//{attribute 'qualified_only'}
VAR_GLOBAL
    (*DP1 ISOLATION VALVE*)
    {attribute 'TcLinkTo' := 	'.i_xOpnLS	:=	TIIB[K4S8_DRL_03_E10_EL1004]^Channel 1^Input;
                                 .i_xClsLS	:=	TIIB[K4S8_DRL_03_E10_EL1004]^Channel 2^Input;
                                 .q_xOPN_DO	:=	TIIB[K4S8_DRL_03_E11_EL2004]^Channel 2^Output
    '}
    {attribute 'pytmc' :=' pv: DREAM:DP1:VRC:01'}
    DREAM_DP1_VRC_01: FB_VRC;

    {attribute 'TcLinkTo' := 	'.i_xOpnLS	:=	TIIB[K4S8_DRL_03_E10_EL1004]^Channel 3^Input;
                                 .i_xClsLS	:=	TIIB[K4S8_DRL_03_E10_EL1004]^Channel 4^Input;
                                 .q_xCLS_DO	:=	TIIB[K4S8_DRL_03_E11_EL2004]^Channel 1^Output
    '}
    {attribute 'pytmc' :=' pv: DREAM:DP1:VRC:02'}
    DREAM_DP1_VRC_02: FB_VRC_NO;

    (*CATCHER 1 ISOLATION VALVE*)
    {attribute 'TcLinkTo' := 	'.i_xOpnLS	:=	TIIB[K4S8_DRL_04_E1_EL1004]^Channel 1^Input;
                                 .i_xClsLS	:=	TIIB[K4S8_DRL_04_E1_EL1004]^Channel 2^Input;
                                 .q_xOPN_DO	:=	TIIB[K4S8_DRL_04_E2_EL2004]^Channel 1^Output
    '}
    {attribute 'pytmc' :=' pv: DREAM:CAT1:VRC:01'}
    DREAM_CAT1_VRC_01: FB_VRC;

    (*ANGLE VALVES ROUGHING*)
    //Pneumatic valves
    {attribute 'TcLinkTo' := 	'.i_xOpnLS	:=	TIIB[K4S8_DRL_04_E9_EL1004]^Channel 1^Input;
                                 .i_xClsLS	:=	TIIB[K4S8_DRL_04_E9_EL1004]^Channel 2^Input;
                                 .q_xOPN_DO	:=	TIIB[K4S8_DRL_04_E11_EL2004]^Channel 1^Output
    '}
    {attribute 'pytmc' :=' pv: DREAM:ROUGH1:VRC:01'}
    DREAM_ROUGH1_VRC_01: FB_VRC; //replacing with VRC function

    {attribute 'TcLinkTo' := 	'.i_xOpnLS	:=	TIIB[K4S8_DRL_04_E9_EL1004]^Channel 3^Input;
                                 .i_xClsLS	:=	TIIB[K4S8_DRL_04_E9_EL1004]^Channel 4^Input;
                                 .q_xOPN_DO	:=	TIIB[K4S8_DRL_04_E11_EL2004]^Channel 2^Output
    '}
    {attribute 'pytmc' :=' pv: DREAM:ROUGH2:VRC:01'}
    DREAM_ROUGH2_VRC_01: FB_VRC; //replacing with VRC function

    {attribute 'TcLinkTo' := 	'.i_xOpnLS	:=	TIIB[K4S8_DRL_04_E10_EL1004]^Channel 1^Input;
                                 .i_xClsLS	:=	TIIB[K4S8_DRL_04_E10_EL1004]^Channel 2^Input;
                                 .q_xOPN_DO	:=	TIIB[K4S8_DRL_04_E11_EL2004]^Channel 3^Output
    '}
    {attribute 'pytmc' :=' pv: DREAM:ROUGH2:VRC:02'}
    DREAM_ROUGH2_VRC_02: FB_VRC; //replacing with VRC function

    (*VENT VALVES ROUGHING*)
    //FLow Control valves MKS248
    {attribute 'TcLinkTo' := 	'.q_iRawPosition	:=	TIIB[WALL_E_PPL_01_EP1_EP4374-0002]^AO Outputs Channel 3^Analog output'}
    {attribute 'pytmc' := 'pv: DREAM:ROUGH1:VFV:01'}
    DREAM_ROUGH1_VFV_01 : FB_MKS248;

    {attribute 'TcLinkTo' := 	'.q_iRawPosition	:=	TIIB[K4S8_DRL_04_EP1_EP4374-0002]^AO Outputs Channel 3^Analog output'}
    {attribute 'pytmc' := 'pv: DREAM:ROUGH1:VFV:02'}
    DREAM_ROUGH1_VFV_02 : FB_MKS248;

    {attribute 'TcLinkTo' := 	'.q_iRawPosition	:=	TIIB[WALL_E_PPL_01_EP1_EP4374-0002]^AO Outputs Channel 4^Analog output'}
    {attribute 'pytmc' := 'pv: DREAM:ROUGH2:VFV:01'}
    DREAM_ROUGH2_VFV_01 : FB_MKS248;

    {attribute 'TcLinkTo' := 	'.q_iRawPosition	:=	TIIB[K4S8_DRL_04_EP1_EP4374-0002]^AO Outputs Channel 4^Analog output'}
    {attribute 'pytmc' := 'pv: DREAM:ROUGH2:VFV:02'}
    DREAM_ROUGH2_VFV_02 : FB_MKS248;

    {attribute 'TcLinkTo' := 	'.q_iRawPosition	:=	TIIB[K4S8_DRL_04_EP2_EP4374-0002]^AO Outputs Channel 3^Analog output'}
    {attribute 'pytmc' := 'pv: DREAM:ROUGH2:VFV:03'}
    DREAM_ROUGH2_VFV_03 : FB_MKS248;

END_VAR

(* stored: Version 1.1.0.1, ProductVersion 3.1.4024.12
   GVL GVL_VAC_VALVES: Id {a72cc40e-50ed-4944-b909-0cce3e1705dc} *)
